{attribute 'conditionalshow'}
TYPE ST_Symbol_Upload_Info :
STRUCT
	{attribute 'hide'}
	udiSymbols				: UDINT;				//Number of symbols on plc
	{attribute 'hide'}
	udiSymbolSize			: UDINT;				//Size of symbols on plc
END_STRUCT
END_TYPE

(* stored: Version 1.1.0.1, ProductVersion 3.1.4024.6
   DUT ST_Symbol_Upload_Info: Id {fde06701-e5c6-4c7b-8314-ee7620a81c2d} *)
